// Mitsubishi GX Works2 project: BookEX6_4 Arithmetric   PLC: Q13UDV

// global labels: Global
VAR_GLOBAL
  bVar0 AT M5000 : BOOL;
  abArray0 AT M5010 : ARRAY [0..49] OF BOOL;
  sStr0 AT D5000 : STRING[199];
  sStr1 AT D5100 : STRING[199];
  sStr2 AT D5200 : STRING[199];
  sStr3 AT D5300 : STRING[199];
  sStr4 AT D5400 : STRING[199];
  sStr5 AT D5500 : STRING[199];
  sStr6 AT D5600 : STRING[199];
  sStr7 AT D5700 : STRING[199];
  sStr8 AT D5800 : STRING[199];
  sStr9 AT D5900 : STRING[199];
  iVar0 AT D4500 : INT;
  iVar1 AT D4501 : INT;
  iVar2 AT D4502 : INT;
  iVar3 AT D4503 : INT;
  iVar4 AT D4504 : INT;
  iVar5 AT D4505 : INT;
  iVar6 AT D4506 : INT;
  iVar7 AT D4507 : INT;
  iVar8 AT D4508 : INT;
  iVar9 AT D4509 : INT;
  dVar0 AT D4510 : DINT;
  dVar1 AT D4512 : DINT;
  dVar2 AT D4514 : DINT;
  dVar3 AT D4516 : DINT;
  dVar4 AT D4518 : DINT;
  dVar5 AT D4520 : DINT;
  dVar6 AT D4522 : DINT;
  dVar7 AT D4524 : DINT;
  dVar8 AT D4526 : DINT;
  dVar9 AT D4528 : DINT;
  wVar0 AT D4530 : WORD;
  wVar1 AT D4531 : WORD;
  wVar2 AT D4532 : WORD;
  wVar3 AT D4533 : WORD;
  wVar4 AT D4534 : WORD;
  wVar5 AT D4535 : WORD;
  wVar6 AT D4536 : WORD;
  wVar7 AT D4537 : WORD;
  wVar8 AT D4538 : WORD;
  wVar9 AT D4539 : WORD;
  dwVar0 AT D4540 : DWORD;
  dwVar1 AT D4542 : DWORD;
  dwVar2 AT D4544 : DWORD;
  dwVar3 AT D4546 : DWORD;
  dwVar4 AT D4548 : DWORD;
  dwVar5 AT D4550 : DWORD;
  dwVar6 AT D4552 : DWORD;
  dwVar7 AT D4554 : DWORD;
  dwVar8 AT D4556 : DWORD;
  dwVar9 AT D4558 : DWORD;
  fsVar0 AT D4560 : REAL;
  fsVar1 AT D4562 : REAL;
  fsVar2 AT D4564 : REAL;
  fsVar3 AT D4566 : REAL;
  fsVar4 AT D4568 : REAL;
  fsVar5 AT D4570 : REAL;
  fsVar6 AT D4572 : REAL;
  fsVar7 AT D4574 : REAL;
  fsVar8 AT D4576 : REAL;
  fsVar9 AT D4578 : REAL;
  fdVar0 AT D4580 : LREAL;
  tTime0 AT D4620 : TIME;
  tTime1 AT D4622 : TIME;
  tTime2 AT D4624 : TIME;
  tTime3 AT D4626 : TIME;
  tTime4 AT D4628 : TIME;
  tTime5 AT D4630 : TIME;
  tTime6 AT D4632 : TIME;
  tTime7 AT D4634 : TIME;
  tTime8 AT D4636 : TIME;
  tTime9 AT D4638 : TIME;
  tTime10 AT D4640 : TIME;
  bVar1 AT M5001 : BOOL;
  bVar2 AT M5002 : BOOL;
  bVar3 AT M5003 : BOOL;
  bVar4 AT M5004 : BOOL;
  bVar5 AT M5005 : BOOL;
  bVar6 AT M5006 : BOOL;
  bVar7 AT M5007 : BOOL;
  bVar8 AT M5008 : BOOL;
  bVar9 AT M5009 : BOOL;
  abArray1 AT M5060 : ARRAY [0..49] OF BOOL;
  abArray2 AT M5110 : ARRAY [0..49] OF BOOL;
  abArray3 AT M5160 : ARRAY [0..49] OF BOOL;
  abArray4 AT M5210 : ARRAY [0..49] OF BOOL;
  abArray5 AT M5260 : ARRAY [0..49] OF BOOL;
  abArray6 AT M5310 : ARRAY [0..49] OF BOOL;
  abArray7 AT M5360 : ARRAY [0..49] OF BOOL;
  abArray8 AT M5410 : ARRAY [0..49] OF BOOL;
  abArray9 AT M5460 : ARRAY [0..49] OF BOOL;
  fdVar1 AT D4584 : LREAL;
  fdVar2 AT D4588 : LREAL;
  fdVar3 AT D4592 : LREAL;
  fdVar4 AT D4596 : LREAL;
  fdVar5 AT D4600 : LREAL;
  fdVar6 AT D4604 : LREAL;
  fdVar7 AT D4608 : LREAL;
  fdVar8 AT D4612 : LREAL;
  fdVar9 AT D4616 : LREAL;
  afsPen0 AT D2000 : ARRAY [0..499] OF REAL;
  afsPen1 AT D3000 : ARRAY [0..499] OF REAL;
END_VAR
// user libraries (not included): HMI

FUNCTION CEIL
VAR_INPUT
  fs_IN : REAL;
END_VAR
VAR
  fsTemp : REAL;
  ix : INT;
END_VAR
;
ix := REAL_TO_INT(fs_IN);
fsTemp := INT_TO_REAL(ix);
IF fsTemp < fs_IN THEN
	ix:= ix+ 1;
END_IF;
CEIL := ix;
END_FUNCTION

FUNCTION_BLOCK DispHMI
VAR_INPUT
  Bit0 : BOOL;
  Bit1 : BOOL;
  Bit3 : BOOL;
  Bit2 : BOOL;
  Bit4 : BOOL;
  Bit5 : BOOL;
  Bit6 : BOOL;
  Bit7 : BOOL;
END_VAR
VAR_OUTPUT
  Data0 : INT;
  Data1 : INT;
  Data2 : INT;
  Data4 : INT;
  Data3 : INT;
  Data5 : INT;
  Data6 : INT;
  Data7 : INT;
END_VAR
(* structured ladder/FBD written out as ST: instructions are called as NAME(EN, inputs, outputs); _pN, _eN, _tN stand for wires *)
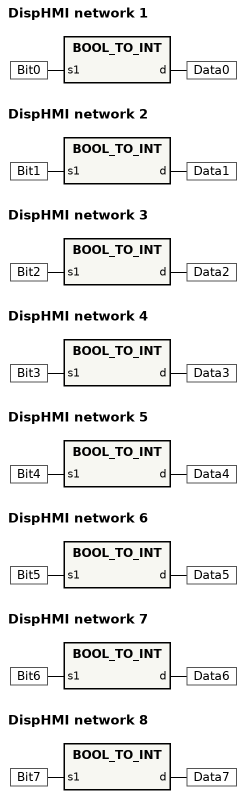
(* network 1 *)
Data0 := BOOL_TO_INT(Bit0);
(* network 2 *)
Data1 := BOOL_TO_INT(Bit1);
(* network 3 *)
Data2 := BOOL_TO_INT(Bit2);
(* network 4 *)
Data3 := BOOL_TO_INT(Bit3);
(* network 5 *)
Data4 := BOOL_TO_INT(Bit4);
(* network 6 *)
Data5 := BOOL_TO_INT(Bit5);
(* network 7 *)
Data6 := BOOL_TO_INT(Bit6);
(* network 8 *)
Data7 := BOOL_TO_INT(Bit7);
END_FUNCTION_BLOCK

FUNCTION_BLOCK DispHMI1
VAR_INPUT
  b_RST : BOOL;
  b_WR : BOOL;
  dw_Data : DWORD;
  b_Data : BOOL;
END_VAR
VAR
  Buffer : ARRAY [0..7] OF WordBit;
  ix : INT;
END_VAR
;
IF LDP(TRUE, b_RST) OR  LDP(TRUE, b_WR) THEN
	IF LDP(TRUE, b_RST) THEN
		FOR ix := 0 TO 7 BY 1 DO
			Buffer[ix].Data := 0;
			Buffer[ix].Flag := FALSE;
		END_FOR;
	ELSE
		FOR ix := 0 TO 6 BY 1 DO
			Buffer[7-ix].Data := Buffer[6-ix].Data; 
			Buffer[7-ix].Flag := Buffer[6-ix].Flag;
		END_FOR;
		Buffer[0].Data := dw_Data;
		Buffer[0].Flag := b_Data;
 	END_IF;
 	FOR ix := 0 TO 7 BY 1 DO
		adwD10[ix] := Buffer[ix].Data; 
		abM10[ix] := Buffer[ix].Flag;
	END_FOR;
END_IF;
END_FUNCTION_BLOCK

FUNCTION_BLOCK DispHMI2
VAR_INPUT
  Str0 : STRING[199];
  Str1 : STRING[199];
  Str2 : STRING[199];
  Str3 : STRING[199];
  Str4 : STRING[199];
  Str5 : STRING[199];
  Str6 : STRING[199];
  Str7 : STRING[199];
  Str8 : STRING[199];
  Str9 : STRING[199];
END_VAR
(* structured ladder/FBD written out as ST: instructions are called as NAME(EN, inputs, outputs); _pN, _eN, _tN stand for wires *)
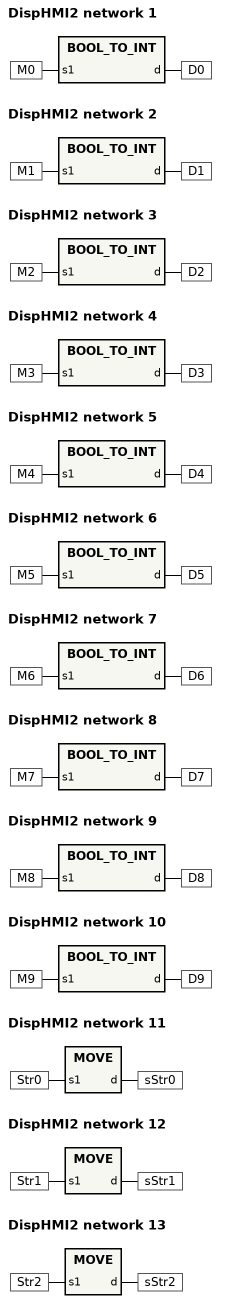
(* network 1 *)
D0 := BOOL_TO_INT(M0);
(* network 2 *)
D1 := BOOL_TO_INT(M1);
(* network 3 *)
D2 := BOOL_TO_INT(M2);
(* network 4 *)
D3 := BOOL_TO_INT(M3);
(* network 5 *)
D4 := BOOL_TO_INT(M4);
(* network 6 *)
D5 := BOOL_TO_INT(M5);
(* network 7 *)
D6 := BOOL_TO_INT(M6);
(* network 8 *)
D7 := BOOL_TO_INT(M7);
(* network 9 *)
D8 := BOOL_TO_INT(M8);
(* network 10 *)
D9 := BOOL_TO_INT(M9);
(* network 11 *)
sStr0 := MOVE(Str0);
(* network 12 *)
sStr1 := MOVE(Str1);
(* network 13 *)
sStr2 := MOVE(Str2);
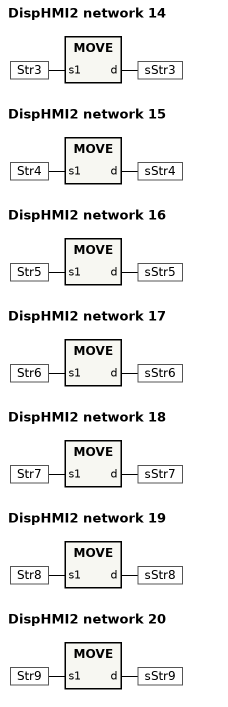
(* network 14 *)
sStr3 := MOVE(Str3);
(* network 15 *)
sStr4 := MOVE(Str4);
(* network 16 *)
sStr5 := MOVE(Str5);
(* network 17 *)
sStr6 := MOVE(Str6);
(* network 18 *)
sStr7 := MOVE(Str7);
(* network 19 *)
sStr8 := MOVE(Str8);
(* network 20 *)
sStr9 := MOVE(Str9);
END_FUNCTION_BLOCK

FUNCTION_BLOCK DIVR
VAR_INPUT
  fs_IN : REAL;
  fs_DIV : REAL;
END_VAR
VAR
  dFloor : DINT;
END_VAR
VAR_OUTPUT
  fs_Q : REAL;
  fs_R : REAL;
END_VAR
VAR
  fsTemp : REAL;
END_VAR
;
IF fs_DIV = 0.0 THEN
	fs_Q := 0.0;
	fs_R := 0.0;
ELSE
	fsTemp := fs_IN / fs_DIV;
	dFloor := REAL_TO_DINT(fsTemp);
	IF DINT_TO_REAL(dFloor) > fsTemp THEN
		dFloor := dFloor - 1;
	END_IF; 
	fs_Q := DINT_TO_REAL(dFloor);
	fs_R := fs_IN - fs_Q * fs_DIV;
END_IF;
END_FUNCTION_BLOCK

FUNCTION FLOOR
VAR_INPUT
  fs_IN : REAL;
END_VAR
VAR
  fsTemp : REAL;
END_VAR
;
FLOOR := REAL_TO_INT(fs_IN);
fsTemp := INT_TO_REAL(FLOOR);
IF fsTemp > fs_IN THEN
	FLOOR := FLOOR - 1;
END_IF;
END_FUNCTION

FUNCTION MODR
VAR_INPUT
  fs_IN : REAL;
  fs_DIV : REAL;
END_VAR
VAR
  dFloor : DINT;
  fsTemp : REAL;
END_VAR
;
IF fs_DIV = 0.0 THEN
	MODR := 0.0;
ELSE
	fsTemp := fs_IN / fs_DIV;
	dFloor := REAL_TO_DINT(fsTemp);
	IF DINT_TO_REAL(dFloor) > fsTemp THEN
		dFloor := dFloor - 1;
	END_IF; 
	MODR := fs_IN - DINT_TO_REAL(dFloor) * fs_DIV;
END_IF;
END_FUNCTION

FUNCTION ROUND
VAR_INPUT
  fs_IN : REAL;
  i_N : INT;
END_VAR
VAR
  fsTemp : REAL;
END_VAR
;
CASE i_N MOD 8 OF
	0 :	fsTemp := 1.0;
	1 : 	fsTemp := 10.0;
	2 : 	fsTemp := 100.0;
	3 : 	fsTemp := 1000.0;
	4 : 	fsTemp := 10000.0;
	5 : 	fsTemp := 100000.0;
	6 : 	fsTemp := 1000000.0;
	7 : 	fsTemp := 10000000.0;
END_CASE;	
ROUND := DINT_TO_REAL(REAL_TO_DINT(fs_IN * fsTemp)) / fsTemp;
END_FUNCTION

FUNCTION_BLOCK Schmitt
VAR_INPUT
  fs_IN : REAL;
  fs_High : REAL;
  fs_Low : REAL;
END_VAR
VAR_OUTPUT
  b_Q : BOOL;
  b_Win : BOOL;
END_VAR
;
IF fs_IN < fs_Low THEN
	b_Q := TRUE;
	b_Win := FALSE;
ELSIF fs_IN > fs_High THEN
	b_Q := FALSE;
	b_Win := FALSE;
ELSE
	b_Win := TRUE;
END_IF;
END_FUNCTION_BLOCK

FUNCTION_BLOCK SM_AVG
VAR_INPUT
  fs_IN : REAL;
END_VAR
VAR_OUTPUT
  fs_Avg : REAL;
  fs_Min : REAL;
END_VAR
VAR
  afsData : ARRAY [0..7] OF REAL;
  DataCnt : INT;
END_VAR
VAR_OUTPUT
  fs_Max : REAL;
END_VAR
VAR_INPUT
  b_EN : BOOL;
  b_Reset : BOOL;
END_VAR
VAR
  ix : INT;
END_VAR
VAR_OUTPUT
  b_ENO : BOOL;
END_VAR
VAR
  fsTemp : REAL;
  fsMin : REAL;
  fsMax : REAL;
END_VAR
;
b_ENO := b_EN;
IF b_Reset THEN
	FOR ix := 0 TO 7 DO
		afsData[ix] := 0.0;
	END_FOR;
	fs_Avg := 0.0;
	fs_Min := 1.0;
	fs_Max := -1.0;
	DataCnt := -1;
ELSIF NOT b_Reset AND b_EN THEN
	DataCnt := DataCnt + 1;
	IF DataCnt = 8 THEN
		FOR ix:= 0 TO 7 DO 
			afsData[ix] := afsData[ix+1];
		END_FOR;
		DataCnt := 7;
	END_IF;
	afsData[DataCnt] := fs_IN;
	IF fs_IN < fsMin THEN fsMin := fs_IN; END_IF;
	IF fs_IN > fsMax THEN fsMax := fs_IN; END_IF;
	fsTemp := 0.0;
	FOR ix := 0 TO DataCnt DO 
		fsTemp := afsData[ix] + fsTemp;
	END_FOR;
	fs_Avg := fsTemp / INT_TO_REAL(DataCnt+1);
	fs_Min := fsMin;
	fs_Max := fsMax;
END_IF;
END_FUNCTION_BLOCK

PROGRAM ExADD
(* structured ladder/FBD written out as ST: instructions are called as NAME(EN, inputs, outputs); _pN, _eN, _tN stand for wires *)
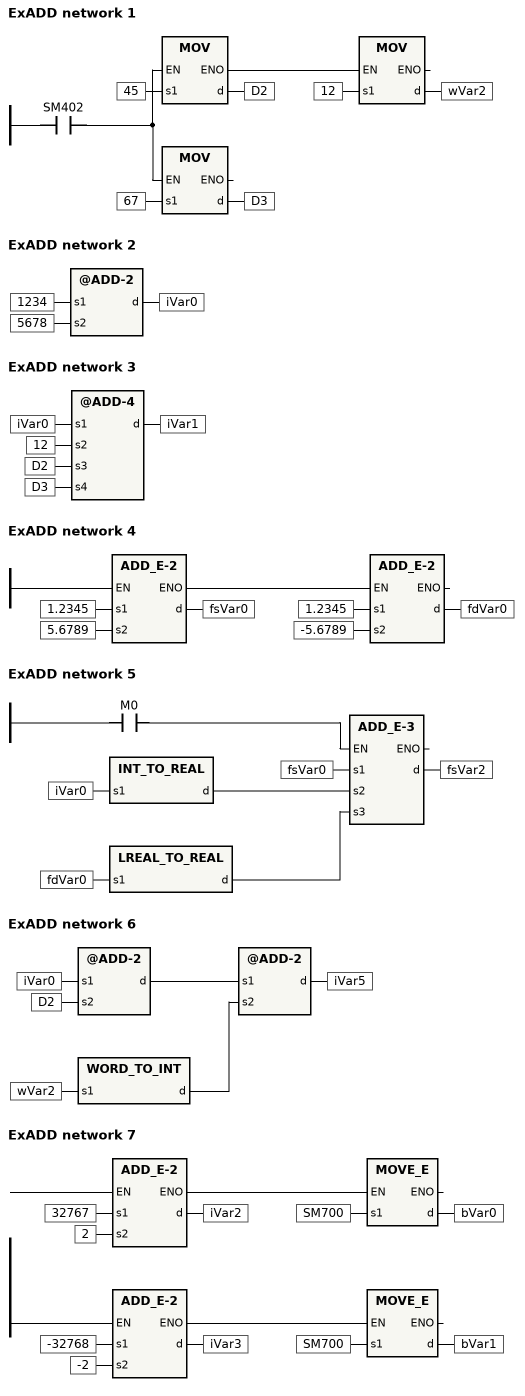
(* network 1 *)
_e1 := MOV(SM402, 45, D2);
MOV(_e1, 12, wVar2);
MOV(SM402, 67, D3);
(* network 2 *)
iVar0 := @ADD-2(1234, 5678);
(* network 3 *)
iVar1 := @ADD-4(iVar0, 12, D2, D3);
(* network 4 *)
_e1 := ADD_E(TRUE, 1.2345, 5.6789, fsVar0);
ADD_E(_e1, 1.2345, -5.6789, fdVar0);
(* network 5 *)
ADD_E(M0, fsVar0, INT_TO_REAL(iVar0), LREAL_TO_REAL(fdVar0), fsVar2);
(* network 6 *)
iVar5 := @ADD-2(@ADD-2(iVar0, D2), WORD_TO_INT(wVar2));
(* network 7 *)
_e1 := ADD_E(TRUE, 32767, 2, iVar2);
MOVE_E(_e1, SM700, bVar0);
_e2 := ADD_E(TRUE, -32768, -2, iVar3);
MOVE_E(_e2, SM700, bVar1);
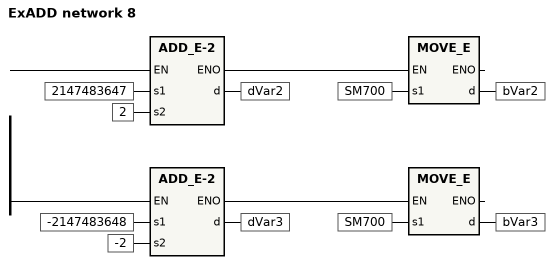
(* network 8 *)
_e1 := ADD_E(TRUE, 2147483647, 2, dVar2);
MOVE_E(_e1, SM700, bVar2);
_e2 := ADD_E(TRUE, -2147483648, -2, dVar3);
MOVE_E(_e2, SM700, bVar3);
END_PROGRAM

PROGRAM ExEXPT
(* structured ladder/FBD written out as ST: instructions are called as NAME(EN, inputs, outputs); _pN, _eN, _tN stand for wires *)
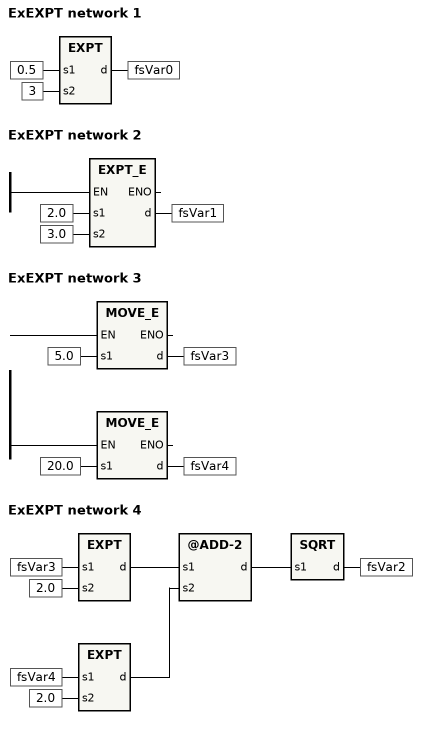
(* network 1 *)
fsVar0 := EXPT(0.5, 3);
(* network 2 *)
EXPT_E(TRUE, 2.0, 3.0, fsVar1);
(* network 3 *)
MOVE_E(TRUE, 5.0, fsVar3);
MOVE_E(TRUE, 20.0, fsVar4);
(* network 4 *)
fsVar2 := SQRT(@ADD-2(EXPT(fsVar3, 2.0), EXPT(fsVar4, 2.0)));
END_PROGRAM

PROGRAM ExMOD
VAR
  DIVR_1 : DIVR;
  fsScale : REAL;
  fsVar : REAL;
  fsQuo : REAL;
  fsResult : REAL;
END_VAR
(* structured ladder/FBD written out as ST: instructions are called as NAME(EN, inputs, outputs); _pN, _eN, _tN stand for wires *)
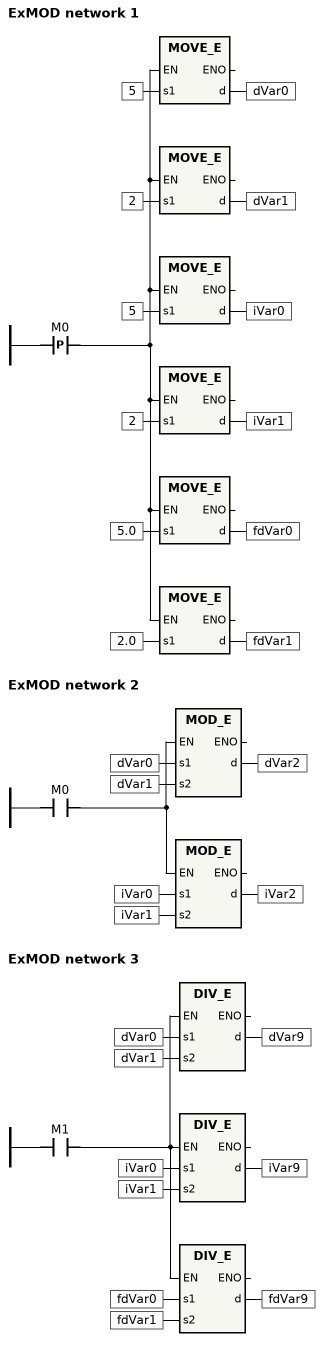
(* network 1 *)
_p1 := LDP(TRUE, M0);
MOVE_E(_p1, 5, dVar0);
MOVE_E(_p1, 2, dVar1);
MOVE_E(_p1, 5, iVar0);
MOVE_E(_p1, 2, iVar1);
MOVE_E(_p1, 5.0, fdVar0);
MOVE_E(_p1, 2.0, fdVar1);
(* network 2 *)
MOD_E(M0, dVar0, dVar1, dVar2);
MOD_E(M0, iVar0, iVar1, iVar2);
(* network 3 *)
DIV_E(M1, dVar0, dVar1, dVar9);
DIV_E(M1, iVar0, iVar1, iVar9);
DIV_E(M1, fdVar0, fdVar1, fdVar9);
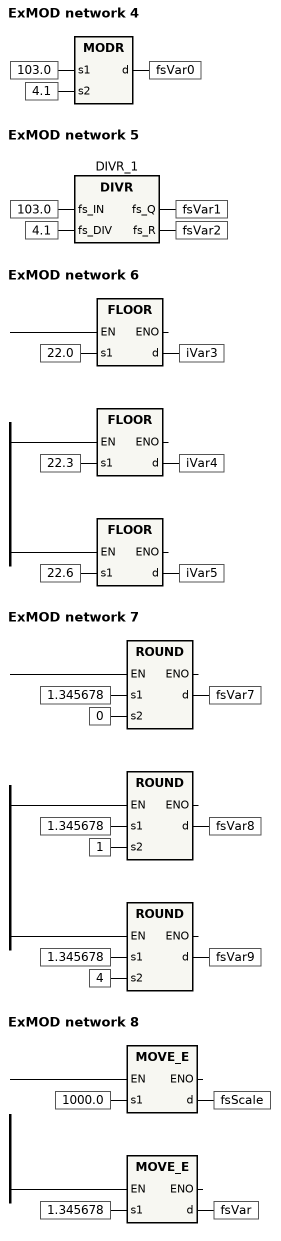
(* network 4 *)
fsVar0 := MODR(103.0, 4.1);
(* network 5 *)
DIVR_1(fs_IN := 103.0, fs_DIV := 4.1, fs_Q => fsVar1, fs_R => fsVar2);
(* network 6 *)
FLOOR(TRUE, 22.0, iVar3);
FLOOR(TRUE, 22.3, iVar4);
FLOOR(TRUE, 22.6, iVar5);
(* network 7 *)
ROUND(TRUE, 1.345678, 0, fsVar7);
ROUND(TRUE, 1.345678, 1, fsVar8);
ROUND(TRUE, 1.345678, 4, fsVar9);
(* network 8 *)
MOVE_E(TRUE, 1000.0, fsScale);
MOVE_E(TRUE, 1.345678, fsVar);
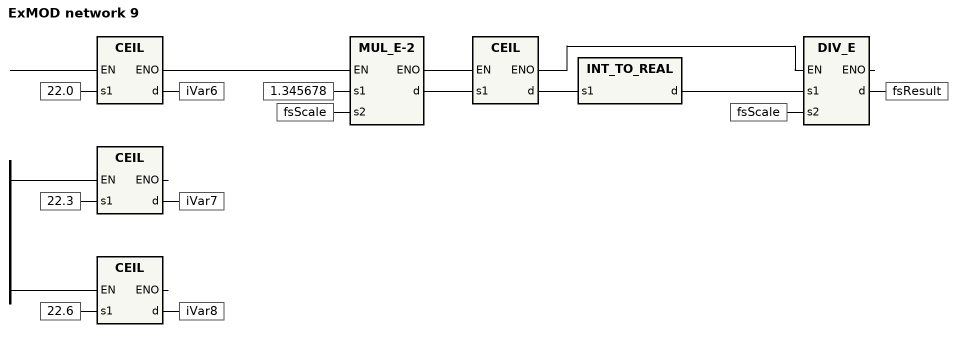
(* network 9 *)
_e1 := CEIL(TRUE, 22.0, iVar6);
_e3 := MUL_E(_e1, 1.345678, fsScale, _t2);
_e5 := CEIL(_e3, _t2, _t4);
CEIL(TRUE, 22.3, iVar7);
DIV_E(_e5, INT_TO_REAL(_t4), fsScale, fsResult);
CEIL(TRUE, 22.6, iVar8);
END_PROGRAM

PROGRAM ExMOD(ST)
;
dVar0 := 5;
dVar1 := 2;
iVar0 := 5;
iVar1 := 2;


dVar2 := dVar0 MOD dVar1;

MOD_E(TRUE, iVar0, iVar1, iVar2);
bVar1 := MOD_E(TRUE, iVar0, iVar1, iVar3);

(*
fsVar4 := 2.0 ** 3;
fsVar2 := EXPT(2.0, 3);
EXPT_E(TRUE, 2.0, 3, fsVar3);
*)
END_PROGRAM

PROGRAM ExMOVE
(* structured ladder/FBD written out as ST: instructions are called as NAME(EN, inputs, outputs); _pN, _eN, _tN stand for wires *)
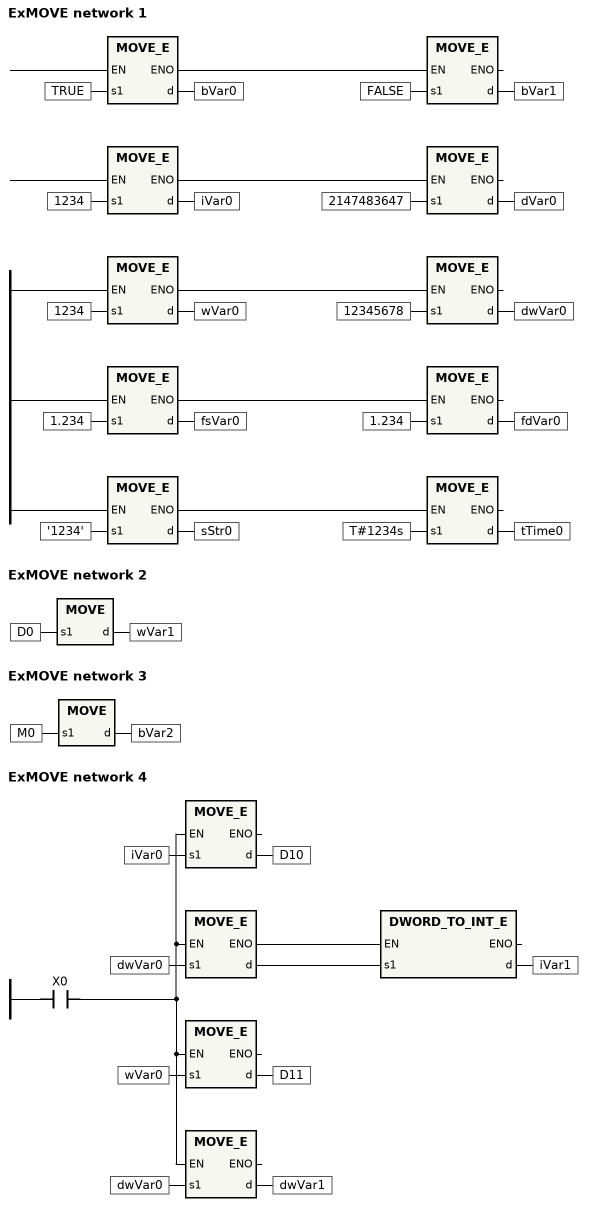
(* network 1 *)
_e1 := MOVE_E(TRUE, TRUE, bVar0);
MOVE_E(_e1, FALSE, bVar1);
_e2 := MOVE_E(TRUE, 1234, iVar0);
MOVE_E(_e2, 2147483647, dVar0);
_e3 := MOVE_E(TRUE, 1234, wVar0);
MOVE_E(_e3, 12345678, dwVar0);
_e4 := MOVE_E(TRUE, 1.234, fsVar0);
MOVE_E(_e4, 1.234, fdVar0);
_e5 := MOVE_E(TRUE, '1234', sStr0);
MOVE_E(_e5, T#1234s, tTime0);
(* network 2 *)
wVar1 := MOVE(D0);
(* network 3 *)
bVar2 := MOVE(M0);
(* network 4 *)
MOVE_E(X0, iVar0, D10);
MOVE_E(X0, wVar0, D11);
MOVE_E(X0, dwVar0, dwVar1);
_e2 := MOVE_E(X0, dwVar0, _t1);
DWORD_TO_INT_E(_e2, _t1, iVar1);
END_PROGRAM

PROGRAM ExMUL
(* structured ladder/FBD written out as ST: instructions are called as NAME(EN, inputs, outputs); _pN, _eN, _tN stand for wires *)
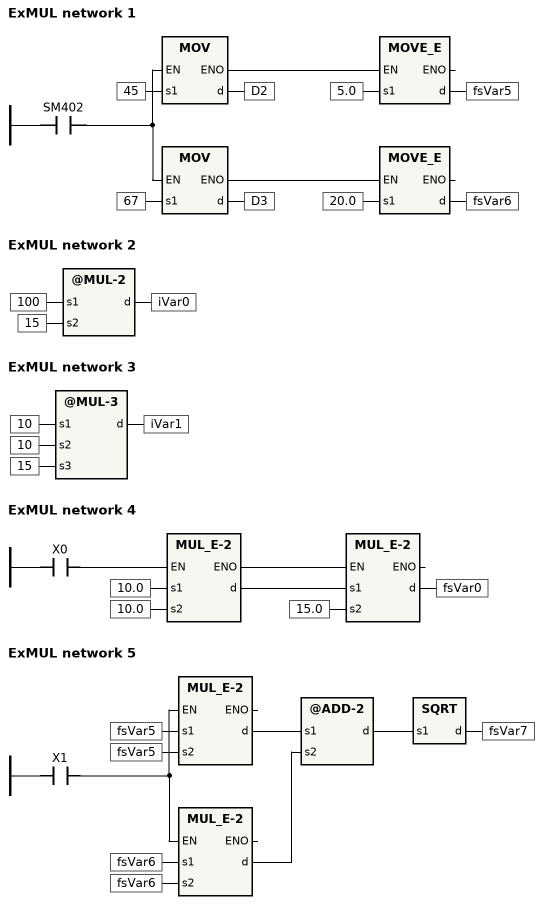
(* network 1 *)
_e1 := MOV(SM402, 45, D2);
MOVE_E(_e1, 5.0, fsVar5);
_e2 := MOV(SM402, 67, D3);
MOVE_E(_e2, 20.0, fsVar6);
(* network 2 *)
iVar0 := @MUL-2(100, 15);
(* network 3 *)
iVar1 := @MUL-3(10, 10, 15);
(* network 4 *)
_e2 := MUL_E(X0, 10.0, 10.0, _t1);
MUL_E(_e2, _t1, 15.0, fsVar0);
(* network 5 *)
MUL_E(X1, fsVar5, fsVar5, _t1);
MUL_E(X1, fsVar6, fsVar6, _t2);
fsVar7 := SQRT(@ADD-2(_t1, _t2));
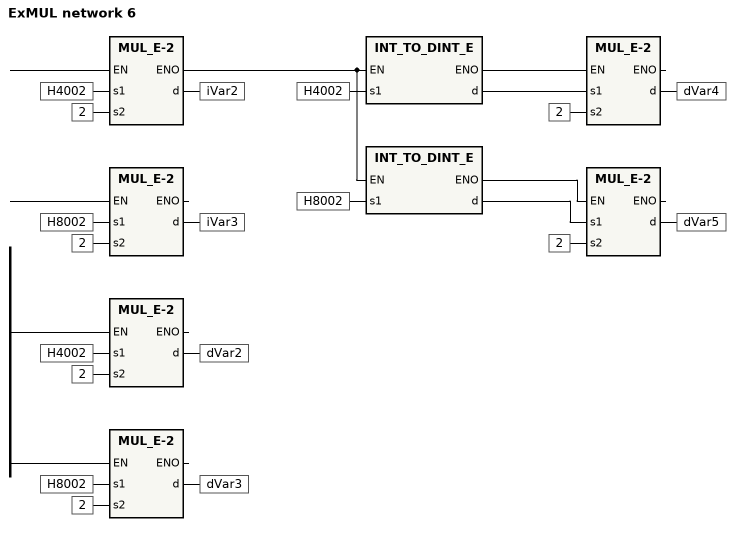
(* network 6 *)
_e1 := MUL_E(TRUE, H4002, 2, iVar2);
_e3 := INT_TO_DINT_E(_e1, H4002, _t2);
MUL_E(_e3, _t2, 2, dVar4);
MUL_E(TRUE, H8002, 2, iVar3);
_e5 := INT_TO_DINT_E(_e1, H8002, _t4);
MUL_E(_e5, _t4, 2, dVar5);
MUL_E(TRUE, H4002, 2, dVar2);
MUL_E(TRUE, H8002, 2, dVar3);
END_PROGRAM

PROGRAM ExSchmitt
VAR
  fbSchmitt : Schmitt;
  ix : INT;
END_VAR
;

IF M2 THEN (* STOP *)
	M0 := FALSE;
	M1 := FALSE;
	iVar0 := 0;
	fsVar0 := 0.0;
	fsVar8 := 1.0;
	fsVar9 := -1.0;
	FOR ix := 0 TO 99 DO 
		afsPen0[ix] := 0.0;
	END_FOR;
	RETURN;
END_IF;

IF M0 THEN (* Up *)
	IF fsVar0 < 0.5 THEN
		fsVar0 := fsVar0 + 0.07;
	ELSE
		fsVar0 := fsVar0 + 0.03;
	END_IF;
	IF fsVar0 > 1.0 THEN 
		fsVar0 := 1.0;
	END_IF;
END_IF;

IF M1 THEN (* Dw *)
	IF fsVar0 < 0.5 THEN
		fsVar0 := fsVar0 - 0.07;
	ELSE
		fsVar0 := fsVar0 - 0.03;
	END_IF;
	IF fsVar0 < 0.0 THEN 
		fsVar0 := 0.0;
	END_IF;
END_IF;
afsPen0[iVar0] := fsVar0;
iVar0 := iVar0 +1;
IF iVar0 > 99 THEN
	iVar0 := 99;
	FOR ix := 1 TO 99 DO 
		afsPen0[ix-1] := afsPen0[ix];
	END_FOR;
END_IF;

fbSchmitt(fs_IN := fsVar0, fs_High := 0.8, fs_Low := 0.6);
M5 := fbSchmitt.b_Q;
M6 := fbSchmitt.b_Win;

IF NOT M5 THEN 
	M0 := FALSE;
	M1 := TRUE;
ELSE
	M0 := TRUE;
	M1 := FALSE;	
END_IF;
END_PROGRAM

PROGRAM ExSM_Avg
VAR
  fbSM_AVG : SM_AVG;
  ix : INT;
  iy : INT;
  iz : INT;
END_VAR
VAR CONSTANT
  cLong : REAL := 0.13;
  cShort : REAL := 0.05;
END_VAR
;

IF M2 THEN (* STOP *)
	M0 := FALSE;
	M1 := FALSE;
	iVar0 := 0;
	fsVar2 := 0.0;
	fsVar8 := 1.0;
	fsVar9 := -1.0;
	FOR ix := 0 TO 359 DO 
		afsPen1[ix] := 0.0;
		afsPen0[ix] := 0.0;
	END_FOR;
	FOR ix := 0 TO 99 DO 
		iy := ix / 10;
		iz := ix MOD 2;
		CASE iy OF 
			0, 1, 8, 9 : (* Inc *)
					IF iz = 0 THEN
						fsVar2 := fsVar2 + cLong;
					ELSE 
						fsVar2 := fsVar2 - cShort;
					END_IF;
			2,7 : (* Hold *)
					IF iz = 0 THEN
						fsVar2 := fsVar2 + cShort;
					ELSE 
						fsVar2 := fsVar2 - cShort;
					END_IF;
			3, 4, 5, 6 : (* Dec *)
					IF iz = 0 THEN
						fsVar2 := fsVar2 - cLong;
					ELSE 
						fsVar2 := fsVar2 + cShort;
					END_IF;
		END_CASE;
		afsPen1[ix*3+3] := fsVar2;
		afsPen1[ix*3+4] := fsVar2;
		afsPen1[ix*3+5] := fsVar2;
	END_FOR;
	fbSM_AVG(b_EN := FALSE, b_Reset := TRUE, fs_IN := 0.0);
	RETURN;
END_IF;

(* IF iVar0 > 2 THEN RETURN; END_IF; *)
	
fbSM_AVG(b_EN := TRUE, b_Reset := FALSE, fs_IN := afsPen1[iVar0]);
afsPen0[iVar0] := fbSM_AVG.fs_Avg;
fsVar0 := fbSM_AVG.fs_Min;
fsVar1 := fbSM_AVG.fs_Max;
iVar0 := iVar0 +1;
IF iVar0 > 359 THEN
	FOR iVar0 := 0 TO 7 DO 
		fbSM_AVG(b_EN := TRUE, b_Reset := FALSE, fs_IN := 0.0);
	END_FOR;
	iVar0 := 0;
END_IF;
END_PROGRAM

PROGRAM ExSUB
(* structured ladder/FBD written out as ST: instructions are called as NAME(EN, inputs, outputs); _pN, _eN, _tN stand for wires *)
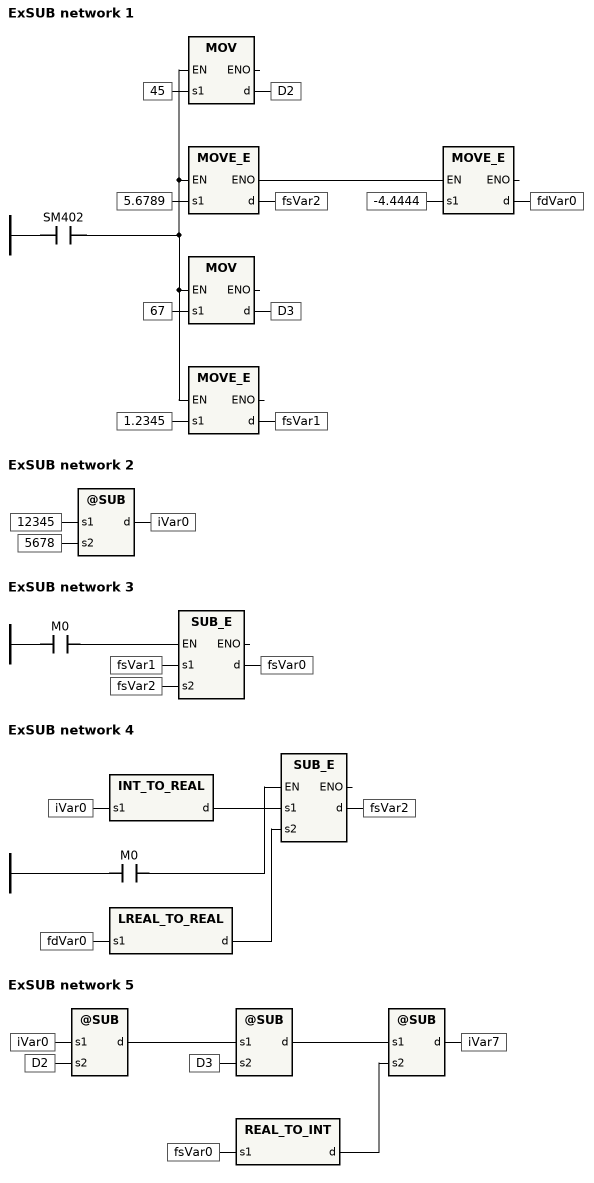
(* network 1 *)
MOV(SM402, 45, D2);
MOV(SM402, 67, D3);
MOVE_E(SM402, 1.2345, fsVar1);
_e1 := MOVE_E(SM402, 5.6789, fsVar2);
MOVE_E(_e1, -4.4444, fdVar0);
(* network 2 *)
iVar0 := @SUB(12345, 5678);
(* network 3 *)
SUB_E(M0, fsVar1, fsVar2, fsVar0);
(* network 4 *)
SUB_E(M0, INT_TO_REAL(iVar0), LREAL_TO_REAL(fdVar0), fsVar2);
(* network 5 *)
iVar7 := @SUB(@SUB(@SUB(iVar0, D2), D3), REAL_TO_INT(fsVar0));
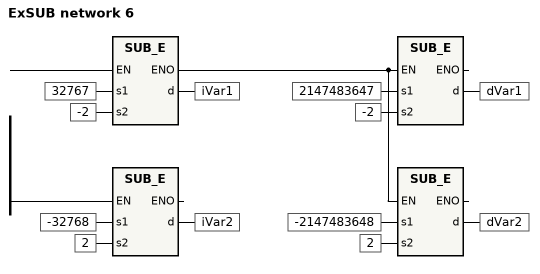
(* network 6 *)
_e1 := SUB_E(TRUE, 32767, -2, iVar1);
SUB_E(_e1, 2147483647, -2, dVar1);
SUB_E(TRUE, -32768, 2, iVar2);
SUB_E(_e1, -2147483648, 2, dVar2);
END_PROGRAM

PROGRAM ExDIV
(* structured ladder/FBD written out as ST: instructions are called as NAME(EN, inputs, outputs); _pN, _eN, _tN stand for wires *)
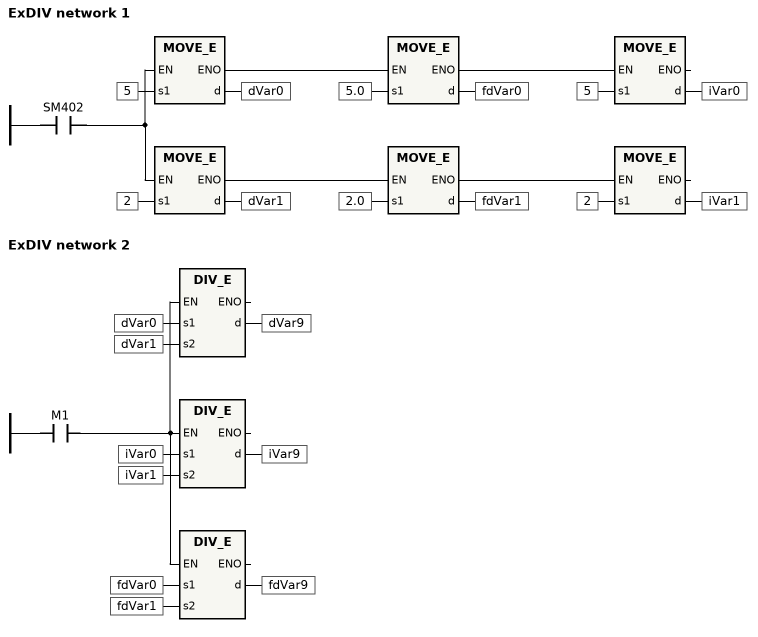
(* network 1 *)
_e1 := MOVE_E(SM402, 5, dVar0);
_e2 := MOVE_E(_e1, 5.0, fdVar0);
MOVE_E(_e2, 5, iVar0);
_e3 := MOVE_E(SM402, 2, dVar1);
_e4 := MOVE_E(_e3, 2.0, fdVar1);
MOVE_E(_e4, 2, iVar1);
(* network 2 *)
DIV_E(M1, dVar0, dVar1, dVar9);
DIV_E(M1, iVar0, iVar1, iVar9);
DIV_E(M1, fdVar0, fdVar1, fdVar9);
END_PROGRAM
